PROGRAM MAIN
VAR
	i :WORD;
END_VAR

i := i +1;

END_PROGRAM

(* stored: Version 1.1.0.1
   POU MAIN: Id {adc68489-9d7f-40b0-9aa9-a9488d4b7fd7}, SpecialFunc None *)
